TYPE ST_CX_EtherCATDeviceState :
STRUCT
	bPresent		: BOOL;
	bOpMode			: BOOL;
	bError			: BOOL;
	nDeviceState	: BYTE;
	nLinkState		: BYTE;
	strStatus		: STRING(17);
END_STRUCT
END_TYPE

(* stored: Version 1.1.0.1, ProductVersion 3.1.4024.15
   DUT ST_CX_EtherCATDeviceState: Id {3860d439-9fa2-42a7-9295-7eeba572a8fc} *)
